% RSLogix 500 project PLC Level 2 Project 5B.RSS, saved by version 8.30.00.16 %
PROJECT "UNTITLED"    % processor: Bul.1763 MicroLogix 1100 Series B %

PROGRAM FILES
  LAD 2   6 rungs

DATA FILES
  O0 OUTPUT  4 elements
  I1 INPUT  6 elements
  S2 STATUS  66 elements
  B3 BINARY  1 elements
  T4 TIMER  2 elements
  C5 COUNTER  1 elements
  R6 CONTROL  1 elements
  N7 INTEGER  1 elements
  F8 FLOAT  3 elements

LADDER 2
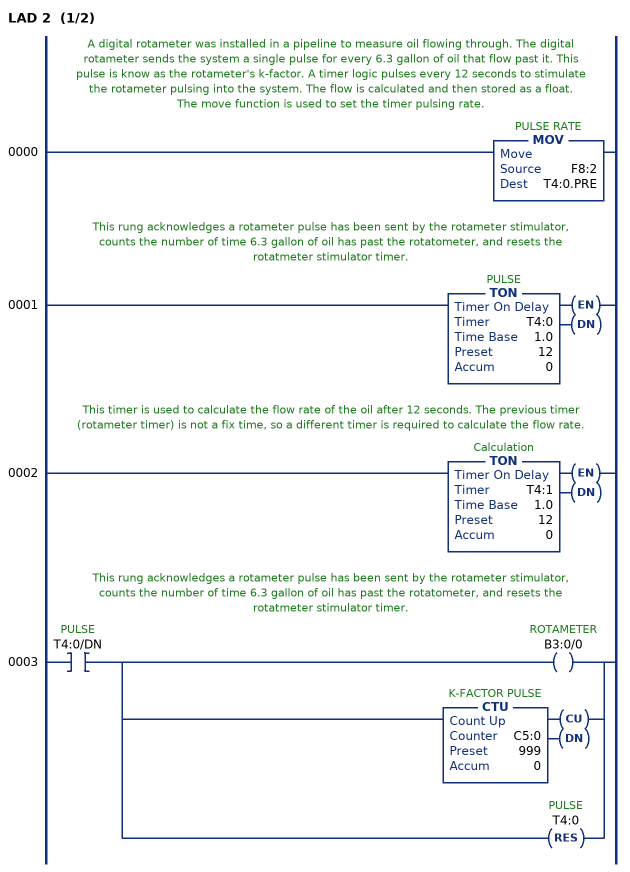
% Rung: 0 %
% A digital rotameter was installed in a pipeline to measure oil flowing through. The digital rotameter sends the system a single pulse for every 6.3 gallon of oil that flow past it. This pulse is know as the rotameter's k-factor. A timer logic pulses every 12 seconds to stimulate the rotameter pulsing into the system. The flow is calculated and then stored as a float.
% The move function is used to set the timer pulsing rate. %
SOR MOV F8:2 T4:0.PRE EOR
%   F8:2  "ARTIFICAL ROTAMETER PULSE" %
%   T4:0.PRE  "PULSE RATE" %
% Rung: 1 %
% This rung acknowledges a rotameter pulse has been sent by the rotameter stimulator, counts the number of time 6.3 gallon of oil has past the rotatometer, and resets the rotatmeter stimulator timer. %
SOR TON T4:0 1.0 12 0 EOR
%   T4:0  "PULSE" %
% Rung: 2 %
% This timer is used to calculate the flow rate of the oil after 12 seconds. The previous timer (rotameter timer) is not a fix time, so a different timer is required to calculate the flow rate. %
SOR TON T4:1 1.0 12 0 EOR
%   T4:1  "Calculation" %
% Rung: 3 %
% This rung acknowledges a rotameter pulse has been sent by the rotameter stimulator, counts the number of time 6.3 gallon of oil has past the rotatometer, and resets the rotatmeter stimulator timer. %
SOR XIC T4:0/DN BST OTE B3:0/0 NXB CTU C5:0 999 0 NXB RES T4:0 BND EOR
%   T4:0/DN  "PULSE" %
%   B3:0/0  "ROTAMETER" %
%   C5:0  "K-FACTOR PULSE" %
%   T4:0  "PULSE" %

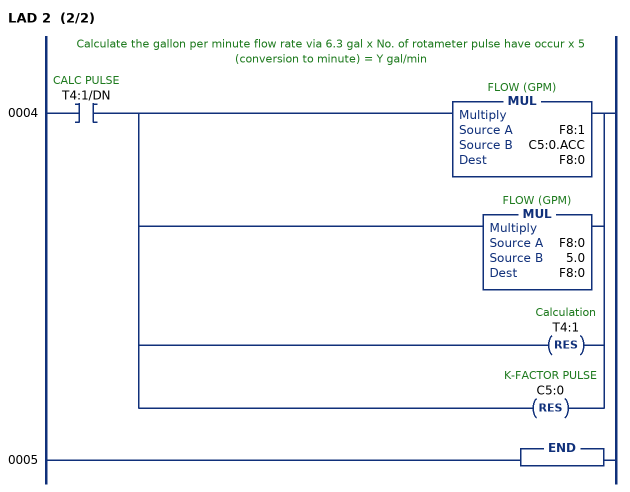
% Rung: 4 %
% Calculate the gallon per minute flow rate via 6.3 gal x No. of rotameter pulse have occur x 5 (conversion to minute) = Y gal/min %
SOR XIC T4:1/DN BST MUL F8:1 C5:0.ACC F8:0 NXB MUL F8:0 5.0 F8:0 NXB RES T4:1 NXB RES C5:0 BND EOR
%   T4:1/DN  "CALC PULSE" %
%   F8:1  "k-factor" %
%   C5:0.ACC  "NUMBER OF K-FACTOR" %
%   F8:0  "FLOW (GPM)" %
%   T4:1  "Calculation" %
%   C5:0  "K-FACTOR PULSE" %
% Rung: 5 %
SOR END EOR

OTHER DOCUMENTED ADDRESSES
  C5:0/DN  "K-FACTOR REST TRIGGER"
  F8:0/1  "k-factor"

DATA TABLE (non-zero values as saved)
DATA T4
% .PRE .ACC %
% T4:0 % 12 0
% T4:1 % 12 0
DATA C5
% .PRE .ACC %
% C5:0 % 999 0
DATA F8
% F8:0 % 0 6.3 12
